Universal Robots PolyScope program: 7_4_pruebas_modbus.urp

Program 7_4_pruebas_modbus (createdIn=3.5.4.10845 lastSavedIn=3.5.4.10845 directory=/programs installation=default robotSerialNumber=2018333608)
Calibrated DH parameters: a=[0.000105, -0.243054, -0.213401, 0.000089, -0.000036, 0]; d=[0.151991, -2.783867, 5.215007, -2.318875, 0.085345, 0.082169]; alpha=[1.572254, -0.00689, -0.001192, 1.571848, -1.571707, 0]; deltaTheta=[-0.000007, 0.078681, -0.09243, 0.013591, 0.000012, 0.000045]
Robot Program (runOnlyOnce=false motionType=MoveJ speed=1.047198 acceleration=1.396263 useActiveTCP=false)
  SuppressedNode
    MoveJ speed 60 deg/s, acceleration 80 deg/s^2 (useActiveTCP=false)
      Waypoint Punto_de_paso_1: TCP in base x=-109.813 y=-299.353 z=126.763 mm, rx=-0.0123 ry=3.1394 rz=0.0018 rad; joints [-90, -90, -90, -90, 90, 0] deg; flange x=-110.206 y=-299.562 z=313.437 mm, rx=-0.0123 ry=3.1395 rz=0.0017 rad
  pose_tcp := get_actual_tcp_pose()
  corrX := read_port_register(128)
  corrY := read_port_register(129)
  pose_corregida := pose_trans(pose_tcp, p[corrX/1000,corrY/1000,0,0,0,0])
  If corrX≠0 or corrY≠0
    If read_port_register(130)≟0
      corrX := -corrX
    If read_port_register(131)≟0
      corrY := -corrY
    MoveL speed 425 mm/s, acceleration 1300 mm/s^2 (useActiveTCP=false) feature=Base
      Waypoint Punto_de_paso (Variable): variable=pose_corregida
  Wait Sleep waitTime=0.01
